{attribute 'linkalways'} 
{attribute 'no_explicit_call' := 'This FB is a CLASS and must be accessed using methods or properties'}
{attribute 'enable_dynamic_creation'}
FUNCTION_BLOCK Node_F_VN_FitLine EXTENDS VisionNode
VAR
    ipPointSet : _ITcVnContainer;
    aFitLine : _TcVnVector4_LREAL;
    hrPrev : _HRESULT(S_OK);
	hresult : _HRESULT(S_OK);
END_VAR

METHOD PUBLIC  Clone : I_Node
VAR
	pNode : POINTER TO Node_F_VN_FitLine;
END_VAR
pNode := __NEW(Node_F_VN_FitLine);
Clone := pNode^;
END_METHOD

METHOD FB_init : BOOL
VAR_INPUT
	bInitRetains : BOOL; // if TRUE, the retain variables are initialized (warm start / cold start)
	bInCopyCode : BOOL;  // if TRUE, the instance afterwards gets moved into the copy code (online change)
END_VAR
AddInput('ipPointSet', ipPointSet);
AddInput('hrPrev', hrPrev);
AddOutput('aFitLine', aFitLine);
AddOutput('hresult',hresult);
END_METHOD

METHOD PROTECTED OnExecute
hresult.Value := F_VN_FitLine(
	ipPointSet := ipPointSet.Value,
    aFitLine := aFitLine.Value,
	hrPrev:= hrPrev.Value);
END_METHOD

METHOD PUBLIC PreExecutionCheck
VAR_INPUT
	Check : I_PreExecutionChecks;
END_VAR
Check.IsTrue(ipPointSet.IsValid, 'ipPointSet must be a valid container');
Check.IsTrue((ipPointSet.IsType(TC_GLOBAL_CONST_LIST.ContainerType_Vector_TcVnPoint2_DINT) OR
              ipPointSet.IsType(TC_GLOBAL_CONST_LIST.ContainerType_Vector_TcVnPoint2_REAL)),
              'ipPointSet contains incorrect type');
END_METHOD

END_FUNCTION_BLOCK

(* stored: Version 1.1.0.1, ProductVersion 3.1.4026.13
   POU Node_F_VN_FitLine: Id {6ca60d88-2c31-0074-1deb-efb0c02f6259}, SpecialFunc None
   Folder Constructor: Id {608b0e60-741b-0168-2c8d-cb3aa139b7b4}
   Method Clone: Id {9bd20a57-3a27-0210-2dd8-f3fbee617574}
   Method FB_init: Id {a6381860-0dbc-06f2-3c48-b4d3163e78f0}
   Method OnExecute: Id {7435ea1f-6f61-03dc-28de-3c60560cebc6}
   Method PreExecutionCheck: Id {99d08ea5-9b3e-08b7-07f3-5acf495a62bc} *)
